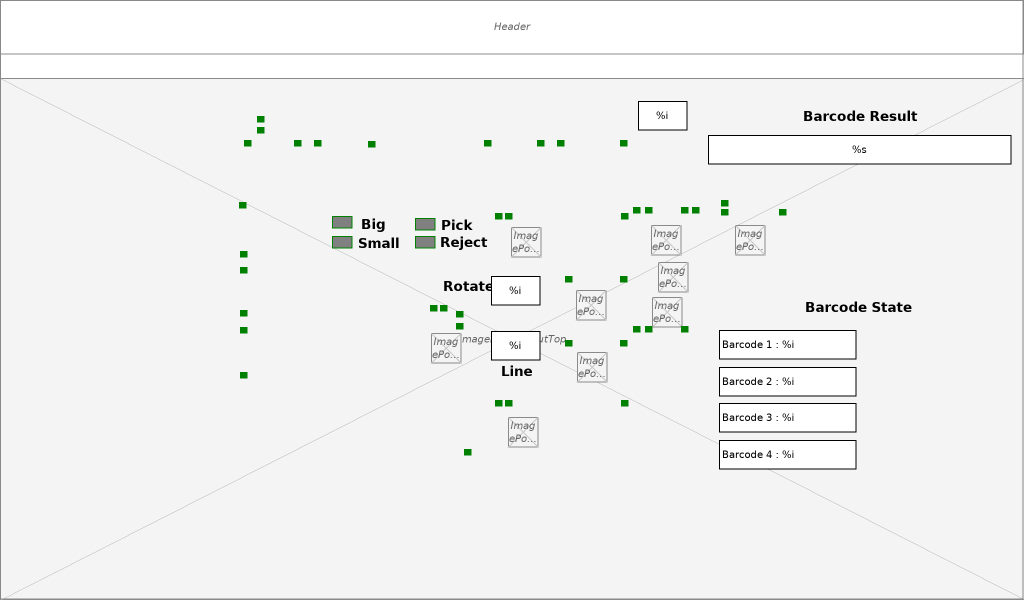
VISUALIZATION SeqStatus  // 1024x600
    Frame (0,-1 1024x55)
        shows Header()
    Label (95,15 250x25), "Machine Status"
    Image (0,78 1026x522), image: ImagePool.LayoutTop
    Image (431,333 30x30), image: ImagePool.info
        OnMouseDown: OpenDialog Dialog=PUSeq, OpenModal=True, OpenCentered=True
        OnMouseDown: execute { HMI_GVL.sCurrentJob :=  HMI_GVL.CJ_Picking; HMI_GVL.iSeqIndex   := HMI_GVL.SI_Picking; }
    Image (511,227 30x30), image: ImagePool.info
        OnMouseDown: OpenDialog Dialog=PUSeq, OpenModal=True, OpenCentered=True
        OnMouseDown: execute { HMI_GVL.sCurrentJob :=  HMI_GVL.CJ_Placing1; HMI_GVL.iSeqIndex   := HMI_GVL.SI_Placing1; }
    Image (576,290 30x30), image: ImagePool.info
        OnMouseDown: OpenDialog Dialog=PUSeq, OpenModal=True, OpenCentered=True
        OnMouseDown: execute { HMI_GVL.sCurrentJob :=  HMI_GVL.CJ_Placing2; HMI_GVL.iSeqIndex   := HMI_GVL.SI_Placing2; }
    Image (577,352 30x30), image: ImagePool.info
        OnMouseDown: OpenDialog Dialog=PUSeq, OpenModal=True, OpenCentered=True
        OnMouseDown: execute { HMI_GVL.sCurrentJob :=  HMI_GVL.CJ_Placing3; HMI_GVL.iSeqIndex   := HMI_GVL.SI_Placing3; }
    Image (508,417 30x30), image: ImagePool.info
        OnMouseDown: OpenDialog Dialog=PUSeq, OpenModal=True, OpenCentered=True
        OnMouseDown: execute { HMI_GVL.sCurrentJob :=  HMI_GVL.CJ_Placing4; HMI_GVL.iSeqIndex   := HMI_GVL.SI_Placing4; }
    Image (735,225 30x30), image: ImagePool.info
        OnMouseDown: OpenDialog Dialog=PUSeq, OpenModal=True, OpenCentered=True
        OnMouseDown: execute { HMI_GVL.sCurrentJob :=  HMI_GVL.CJ_Dispenser; HMI_GVL.iSeqIndex   := InputOutput_GVL.SeqIndexOutfeed[4]; }
    Image (652,297 30x30), image: ImagePool.info
        OnMouseDown: OpenDialog Dialog=PUSeq, OpenModal=True, OpenCentered=True
        OnMouseDown: execute { HMI_GVL.sCurrentJob :=  HMI_GVL.CJ_ShuttleEmpty; HMI_GVL.iSeqIndex   := InputOutput_GVL.SeqIndexOutfeed[1]; }
    Image (651,225 30x30), image: ImagePool.info
        OnMouseDown: OpenDialog Dialog=PUSeq, OpenModal=True, OpenCentered=True
        OnMouseDown: execute { HMI_GVL.sCurrentJob :=  HMI_GVL.CJ_ShuttleLoad; HMI_GVL.iSeqIndex   := InputOutput_GVL.SeqIndexOutfeed[2]; }
    Image (658,262 30x30), image: ImagePool.info
        OnMouseDown: OpenDialog Dialog=PUSeq, OpenModal=True, OpenCentered=True
        OnMouseDown: execute { HMI_GVL.sCurrentJob :=  HMI_GVL.CJ_ShuttleManagement; HMI_GVL.iSeqIndex   := InputOutput_GVL.SeqIndexOutfeed[3]; }
    Rectangle (415,218 20x12), colour toggle: InputOutput_GVL.xOut_Robot.Pick
    Rectangle (415,236 20x12), colour toggle: InputOutput_GVL.xOut_Robot.RejectBox
    Label (438,213 65x25), "Pick"
    Label (437,230 65x25), "Reject"
    Rectangle (456,323 7x6), colour toggle: InputOutput_GVL.xIn1405
    Rectangle (456,311 7x6), colour toggle: InputOutput_GVL.xIn1406
    Rectangle (430,305 7x6), colour toggle: InputOutput_GVL.xIn1407
    Rectangle (440,305 7x6), colour toggle: InputOutput_GVL.xIn1400
    Rectangle (633,207 7x6), colour toggle: InputOutput_GVL.Digital_Input[124]
    Rectangle (645,207 7x6), colour toggle: InputOutput_GVL.Digital_Input[122]
    Rectangle (681,207 7x6), colour toggle: InputOutput_GVL.Digital_Input[121]
    Rectangle (692,207 7x6), colour toggle: InputOutput_GVL.Digital_Input[123]
    Rectangle (633,326 7x6), colour toggle: InputOutput_GVL.Digital_Input[119]
    Rectangle (645,326 7x6), colour toggle: InputOutput_GVL.Digital_Input[117]
    Rectangle (681,326 7x6), colour toggle: InputOutput_GVL.Digital_Input[118]
    Rectangle (721,209 7x6), colour toggle: InputOutput_GVL.Digital_Input[51]
    Rectangle (721,200 7x6), colour toggle: InputOutput_GVL.Digital_Input[52]
    Rectangle (779,209 7x6), colour toggle: InputOutput_GVL.Digital_Input[50]
    Rectangle (495,400 7x6), colour toggle: InputOutput_GVL.xIn1509
    Rectangle (505,400 7x6), colour toggle: InputOutput_GVL.xIn1508
    Rectangle (621,400 7x6), colour toggle: InputOutput_GVL.xIn1507
    Rectangle (565,340 7x6), colour toggle: InputOutput_GVL.xIn1506
    Rectangle (620,340 7x6), colour toggle: InputOutput_GVL.xIn1505
    Rectangle (565,276 7x6), colour toggle: InputOutput_GVL.xIn1504
    Rectangle (620,276 7x6), colour toggle: InputOutput_GVL.xIn1503
    Rectangle (495,213 7x6), colour toggle: InputOutput_GVL.xIn1502
    Rectangle (505,213 7x6), colour toggle: InputOutput_GVL.xIn1501
    Rectangle (621,213 7x6), colour toggle: InputOutput_GVL.xIn1500
    Rectangle (620,140 7x6), colour toggle: InputOutput_GVL.Digital_Input[14]
    Rectangle (557,140 7x6), colour toggle: InputOutput_GVL.Digital_Input[15]
    Rectangle (537,140 7x6), colour toggle: InputOutput_GVL.Digital_Input[37]
    Rectangle (484,140 7x6), colour toggle: InputOutput_GVL.Digital_Input[38]
    Rectangle (368,141 7x6), colour toggle: InputOutput_GVL.Digital_Input[39]
    Rectangle (314,140 7x6), colour toggle: InputOutput_GVL.Digital_Input[40]
    Rectangle (294,140 7x6), colour toggle: InputOutput_GVL.Digital_Input[41]
    Rectangle (244,140 7x6), colour toggle: InputOutput_GVL.Digital_Input[42]
    Rectangle (239,202 7x6), colour toggle: InputOutput_GVL.Digital_Input[45]
    Rectangle (240,251 7x6), colour toggle: InputOutput_GVL.Digital_Input[46]
    Rectangle (240,267 7x6), colour toggle: InputOutput_GVL.Digital_Input[47]
    Rectangle (240,310 7x6), colour toggle: InputOutput_GVL.Digital_Input[48]
    Rectangle (240,327 7x6), colour toggle: InputOutput_GVL.Digital_Input[8]
    Rectangle (240,372 7x6), colour toggle: InputOutput_GVL.Digital_Input[9]
    Rectangle (257,127 7x6), colour toggle: InputOutput_GVL.Digital_Input[43]
    Rectangle (257,116 7x6), colour toggle: InputOutput_GVL.Digital_Input[44]
    Rectangle (464,449 7x6), colour toggle: InputOutput_GVL.xIn1005
    RoundedRectangle (638,101 49x29), "%i", text variable: InputOutput_GVL.ShuttlePosition
    Rectangle (332,216 20x12), colour toggle: InputOutput_GVL.xOut_Robot.CheckBigBox
    Label (358,212 65x25), "Big"
    Rectangle (332,236 20x12), colour toggle: InputOutput_GVL.xOut_Robot.CheckSmallBox
    Label (355,231 65x25), "Small"
    RoundedRectangle (708,135 303x29), "%s", text variable: Status_GVL.BarcodeResult
    Label (712,104 297x25), "Barcode Result"
    Label (710,295 297x25), "Barcode State"
    RoundedRectangle (719,330 137x29), "Barcode 1 : %i", text variable: InputOutput_GVL.BarcodeReader_Picking1_State
    RoundedRectangle (719,367 137x29), "Barcode 2 : %i", text variable: InputOutput_GVL.BarcodeReader_Picking2B_State
    RoundedRectangle (719,403 137x29), "Barcode 3 : %i", text variable: InputOutput_GVL.BarcodeReader_Picking3B_State
    RoundedRectangle (719,440 137x29), "Barcode 4 : %i", text variable: InputOutput_GVL.BarcodeReader_Picking4_State
    RoundedRectangle (491,331 49x29), "%i", text variable: HMI_GVL.PickLine
    Label (440,274 65x25), "Rotate"
    RoundedRectangle (491,276 49x29), "%i", text variable: InputOutput_GVL.xOut_Robot.RotatePickInt
    Label (498,359 65x25), "Line"
END_VISUALIZATION

(* stored: Version 1.1.0.1, ProductVersion 3.1.4024.12
   Visu SeqStatus: Id {75ae1ae9-be1e-4df0-b502-68ef5f65f0de} *)
